DATA_BLOCK "PN-OUTPUT-robot"
{ S7_Optimized_Access := 'FALSE' }
VERSION : 0.1
   STRUCT
      "00" : Byte;   // Заглушка
      a1 : Byte;   // 1DI_BYTE1 датчики захвата
      b1 : Byte;   // 1DI_BYTE2 датчики паллет
      c1 : Byte;   // 1DI_BYTE3 присоски
      d1 : Byte;   // 1DI_BYTE4 UI
      e1 : Byte;   // 1DI_BYTE5 Скорость робота
      f1 : Byte;   // 1
      g1 : Byte;   // 1
      K1 : DWord;   // 1
      O1 : DWord;   // 1
      P1 : Byte;   // RTK1-----------------------
      a2 : Byte;   // 2DI_BYTE1 датчики захвата
      b2 : Byte;   // 2DI_BYTE2 датчики паллет
      c2 : Byte;   // 2DI_BYTE3 присоски
      d2 : Byte;   // 2DI_BYTE4 UI
      e2 : Byte;   // 2DI_BYTE5 Скорость робота
      f2 : Byte;   // 2
      g2 : Byte;   // 2
      N2 : DWord;   // 2
      O2 : DWord;   // 2
      P2 : Byte;   // RTK2-----------------------------
      a3 : Byte;   // 3DI_BYTE1 датчики захвата
      b3 : Byte;   // 3DI_BYTE2 датчики паллет
      c3 : Byte;   // 3DI_BYTE3 присоски
      d3 : Byte;   // 3DI_BYTE4 UI
      e3 : Byte;   // 3DI_BYTE5 Скорость робота
      f3 : Byte;   // 3
      g3 : Byte;   // 3
      N3 : DWord;   // 3
      O3 : DWord;   // 3
      P3 : Byte;   // RTK3--------------------------------
      a4 : Byte;   // 4DI_BYTE1 датчики захвата
      b4 : Byte;   // 4DI_BYTE2 датчики паллет
      c4 : Byte;   // 4DI_BYTE3 присоски
      d4 : Byte;   // 4DI_BYTE4 UI
      e4 : Byte;   // 4DI_BYTE5 Скорость робота
      f4 : Byte;   // 4
      g4 : Byte;   // 4
      N4 : DWord;   // 4
      O4 : DWord;   // 4
      P4 : Byte;   // RTK4
      a7 : Byte;   // заглушка четности
      c7 : DWord;   // FA1------------------------------------------------
      g7 : DWord;   // FA1
      K7 : Word;   // FA1_1_ETA
      a8 : Word;   // FA1_1_Speed
      b7 : DWord;   // FA2------------------------------------------------------
      c8 : DWord;   // FA2
      d7 : Word;   // FA2_1_ETA
      e7 : Word;   // FA2_1_Speed
      f7 : DWord;   // FA3------------------------------------------------
      g8 : DWord;   // FA3
      h7 : Word;   // FA3_1_ETA
      i7 : Word;   // FA3_1_Speed
      J7 : DWord;   // FA23------------------------------------------------------
      K8 : DWord;   // FA23
      L7 : Word;   // FA23_1_ETA
      M5 : Word;   // FA23_1_Speed
      c9 : DWord;   // FA24------------------------------------------------
      g9 : DWord;   // FA24
      K9 : Word;   // FA24_1_ETA
      a9 : Word;   // FA24_1_Speed
      b8 : DWord;   // FA4------------------------------------------------------
      c10 : DWord;   // FA4
      d8 : Word;   // FA4_1_ETA
      e8 : Word;   // FA4_1_Speed
      f8 : DWord;   // FA5------------------------------------------------
      g10 : DWord;   // FA5
      h8 : Word;   // FA5_1_ETA
      i8 : Word;   // FA5_1_Speed
      J8 : DWord;   // FA20------------------------------------------------------
      K10 : DWord;   // FA20
      L8 : Word;   // FA20_1_ETA
      M6 : Word;   // FA20_1_Speed
      c11 : DWord;   // FA25_1------------------------------------------------
      g11 : DWord;   // FA25_1
      K11 : Word;   // FA25_1_ETA
      a10 : Word;   // FA25_1_Speed
      b9 : DWord;   // FA25_2------------------------------------------------------
      c12 : DWord;   // FA25_2
      d9 : Word;   // FA25_2_ETA
      e9 : Word;   // FA25_2_Speed
      f9 : DWord;   // FA6------------------------------------------------
      g12 : DWord;   // FA6
      h9 : Word;   // FA6_1_ETA
      i9 : Word;   // FA6_1_Speed
      J9 : DWord;   // FA7------------------------------------------------------
      K12 : DWord;   // FA7
      L9 : Word;   // FA7_1_ETA
      M7 : Word;   // FA7_1_Speed
      c13 : DWord;   // FA8------------------------------------------------
      g13 : DWord;   // FA8
      K13 : Word;   // FA8_1_ETA
      a11 : Word;   // FA8_1_Speed
      b10 : DWord;   // FA26------------------------------------------------------
      c14 : DWord;   // FA26
      d10 : Word;   // FA26_1_ETA
      e10 : Word;   // FA26_1_Speed
      f10 : DWord;   // FA27------------------------------------------------
      g14 : DWord;   // FA27
      h10 : Word;   // FA27_1_ETA
      i10 : Word;   // FA27_1_Speed
      J10 : DWord;   // FA9------------------------------------------------------
      K14 : DWord;   // FA9
      L10 : Word;   // FA9_1_ETA
      M8 : Word;   // FA9_1_Speed
      J11 : DWord;   // FA10------------------------------------------------------
      K15 : DWord;   // FA10
      L11 : Word;   // FA10_1_ETA
      M9 : Word;   // FA10_1_Speed
      f11 : DWord;   // FA28------------------------------------------------
      g15 : DWord;   // FA28
      h11 : Word;   // FA28_1_ETA
      i11 : Word;   // FA28_1_Speed
      N5 : Word;
      O5 : Word;
      temp_1 : DWord;
      temp3 : DWord;
      temp4 : DWord;
   END_STRUCT;


BEGIN

END_DATA_BLOCK

